Omron Sysmac Studio project Motor_Calisma_Suresi (Sysmac Studio 1.65.0.64007, StandardProject)

# Controller new_Controller_0: NX1P2-1040DT1 version 1.69
Task PrimaryTask (priority 4, period or condition 2000): Program0

VAR_GLOBAL
    Motor : BOOL;
END_VAR
VAR_GLOBAL RETAIN
    CalismaSu : DINT;
    AccT_ET : TIME;
END_VAR
VAR_GLOBAL
    AccT1_ET : TIME;  (* SANİYE *)
    AccT2_ET : TIME;
END_VAR
VAR_GLOBAL RETAIN
    CalismaSure2 : DINT;  (* SAAT *)
    CalismaSure1 : DINT;  (* DAKİKA *)
END_VAR

PROGRAM Program0
VAR
    StartButton : BOOL;
    StopButton : BOOL;
    Start : BOOL;
    AccT1 : AccumulationTimer;
    AccT1_Reset : BOOL;
    Sifir : DINT;
END_VAR
VAR_EXTERNAL
    Motor : BOOL;
    AccT1_ET : TIME;
    CalismaSure2 : DINT;
    CalismaSure1 : DINT;
END_VAR
VAR
    _e1 : R_TRIG;
    _p2 : BOOL;
END_VAR

(* Section Section0: ladder, written here as Structured Text *)

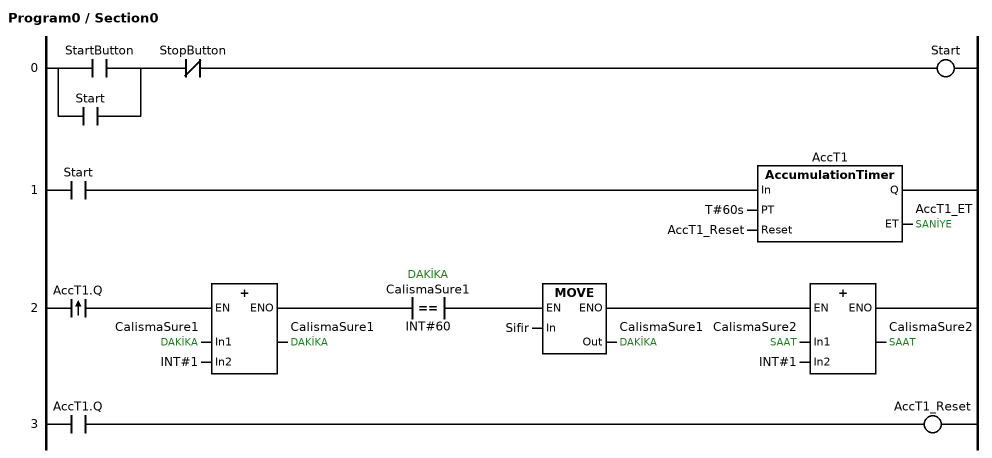
(* Rung 0 *)
Start := (StartButton OR Start) AND NOT StopButton;
(* Rung 1 *)
AccT1(In := Start, PT := T#60s, Reset := AccT1_Reset, ET => AccT1_ET);
(* Rung 2 *)
_e1(CLK := AccT1.Q);
IF _e1.Q THEN CalismaSure1 := CalismaSure1 + INT#1; END_IF;
_p2 := _e1.Q AND (CalismaSure1 = INT#60);
IF _p2 THEN
    CalismaSure1 := Sifir;
    CalismaSure2 := CalismaSure2 + INT#1;
END_IF;
(* Rung 3 *)
AccT1_Reset := AccT1.Q;
END_PROGRAM